PROGRAM Test
VAR
	EdgeD: R_TRIG;
	RS_0: RS;
	CTU_0: CTUD;
	COUNT: CTUD;
	testVar1 : WORD := 11;
	testVar2 : WORD := 0;
	testVar3 : WORD := 12;
		testVar4 : BOOL := TRUE;
		TP_0: TP;
	testVar5 : TIME := T#0ms;
	LEDUBlue: BOOL;
	ms: TIME;
	T1: TON;
	TOF_0: TOF;
	LLBButton: BOOL;
	LED: MotorControla;
	MotorControla_0: MotorControla;
	MotorControla_1: MotorControla;
	MotorControla_2: MotorControla;
	MX: Multiplex;
	Patch: MotorControla;
	MotorControla_3: MotorControla;
	MotorControla_4: MotorControla;
	MotorControla_5: MotorControla;
	IntLck: BOOL;
	IntLck1: BOOL;
	IntLck2: BOOL;
	IntLck3: BOOL;
	Stp3: BOOL;
	Stp1: BOOL;
	Stp2: BOOL;
	Stp4: BOOL;
	Counter_0: Counter;
	KDP: BOOL;
	IntLck4: BOOL;
END_VAR

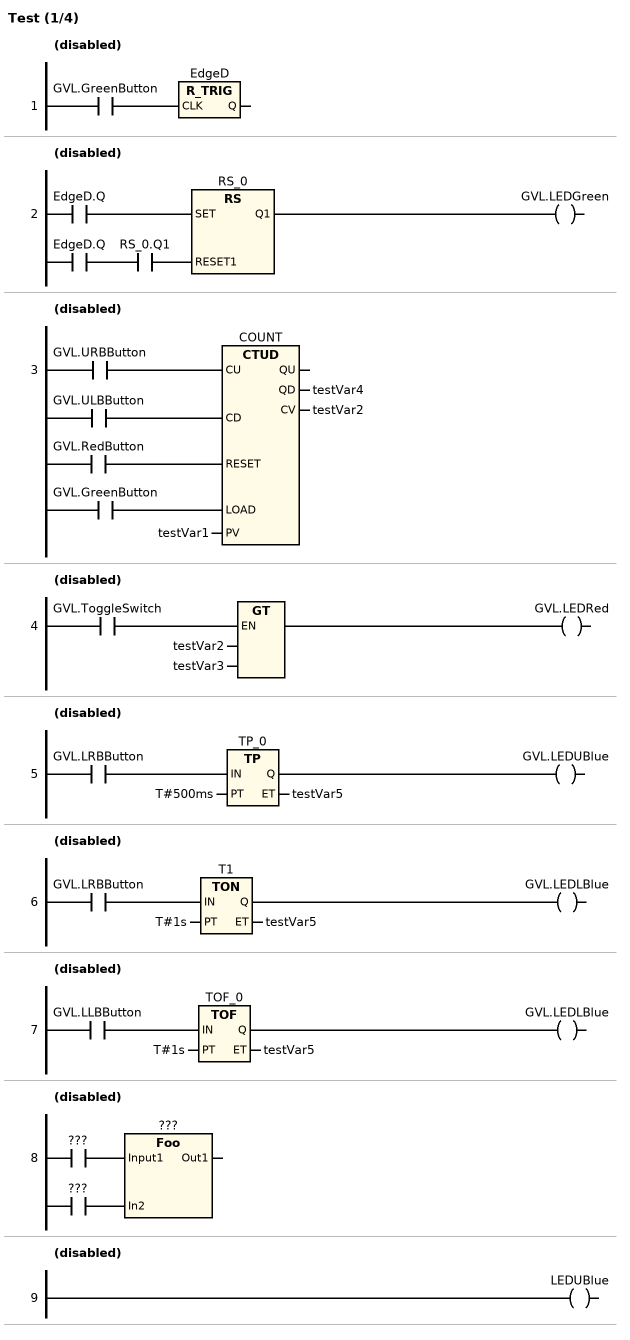
// NETWORK 1 (disabled)
// EdgeD(CLK := GVL.GreenButton); // R_TRIG

// NETWORK 2 (disabled)
// RS_0(SET := EdgeD.Q, RESET1 := EdgeD.Q AND RS_0.Q1); // RS
// GVL.LEDGreen := RS_0.Q1;

// NETWORK 3 (disabled)
// COUNT(
//     CU := GVL.URBButton,
//     CD := GVL.ULBButton,
//     RESET := GVL.RedButton,
//     LOAD := GVL.GreenButton,
//     PV := testVar1,
//     QD => testVar4,
//     CV => testVar2); // CTUD

// NETWORK 4 (disabled)
// GVL.LEDRed := GVL.ToggleSwitch AND testVar2 > testVar3;

// NETWORK 5 (disabled)
// TP_0(IN := GVL.LRBButton, PT := T#500ms, ET => testVar5); // TP
// GVL.LEDUBlue := TP_0.Q;

// NETWORK 6 (disabled)
// T1(IN := GVL.LRBButton, PT := T#1s, ET => testVar5); // TON
// GVL.LEDLBlue := T1.Q;

// NETWORK 7 (disabled)
// TOF_0(IN := GVL.LLBButton, PT := T#1s, ET => testVar5); // TOF
// GVL.LEDLBlue := TOF_0.Q;

// NETWORK 8 (disabled)
// ???(); // Foo

// NETWORK 9 (disabled)
// LEDUBlue := TRUE;

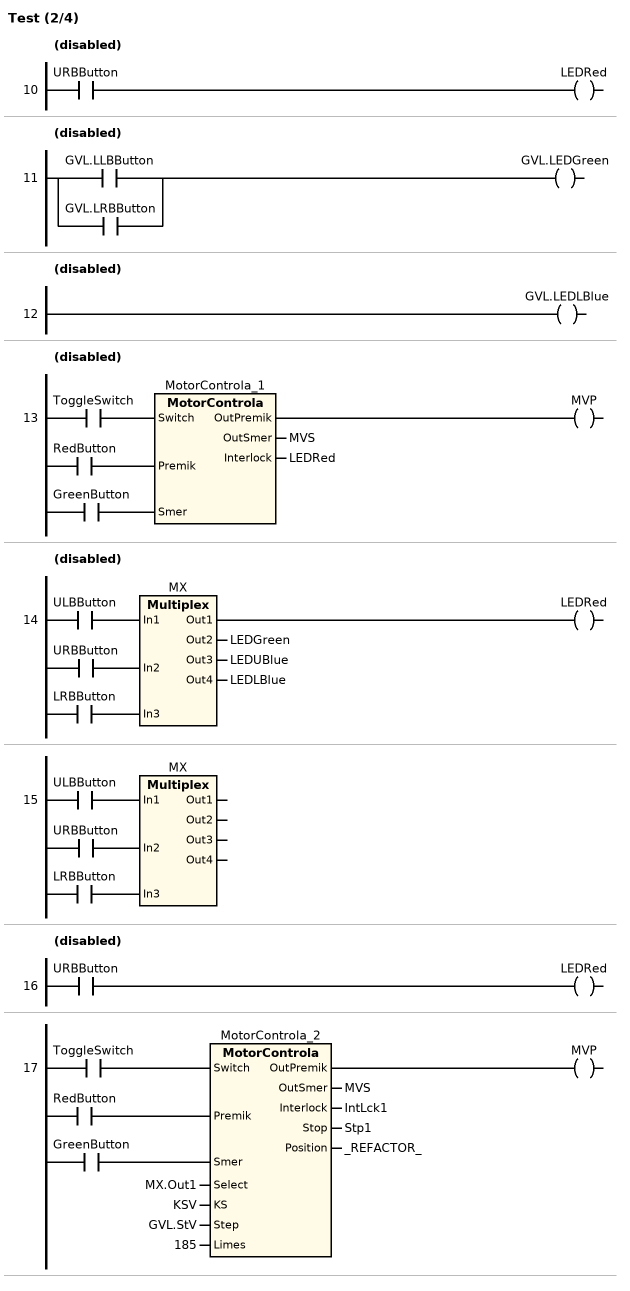
// NETWORK 10 (disabled)
// LEDRed := URBButton;

// NETWORK 11 (disabled)
// GVL.LEDGreen := GVL.LLBButton OR GVL.LRBButton;

// NETWORK 12 (disabled)
// GVL.LEDLBlue := TRUE;

// NETWORK 13 (disabled)
// MotorControla_1(
//     Switch := ToggleSwitch,
//     Premik := RedButton,
//     Smer := GreenButton,
//     OutSmer => MVS,
//     Interlock => LEDRed); // MotorControla
// MVP := MotorControla_1.OutPremik;

// NETWORK 14 (disabled)
// MX(
//     In1 := ULBButton,
//     In2 := URBButton,
//     In3 := LRBButton,
//     Out2 => LEDGreen,
//     Out3 => LEDUBlue,
//     Out4 => LEDLBlue); // Multiplex
// LEDRed := MX.Out1;

// NETWORK 15
MX(In1 := ULBButton, In2 := URBButton, In3 := LRBButton); // Multiplex

// NETWORK 16 (disabled)
// LEDRed := URBButton;

// NETWORK 17
MotorControla_2(
    Switch := ToggleSwitch,
    Premik := RedButton,
    Smer := GreenButton,
    Select := MX.Out1,
    KS := KSV,
    Step := GVL.StV,
    Limes := 185,
    OutSmer => MVS,
    Interlock => IntLck1,
    Stop => Stp1,
    Position => _REFACTOR_); // MotorControla
MVP := MotorControla_2.OutPremik;

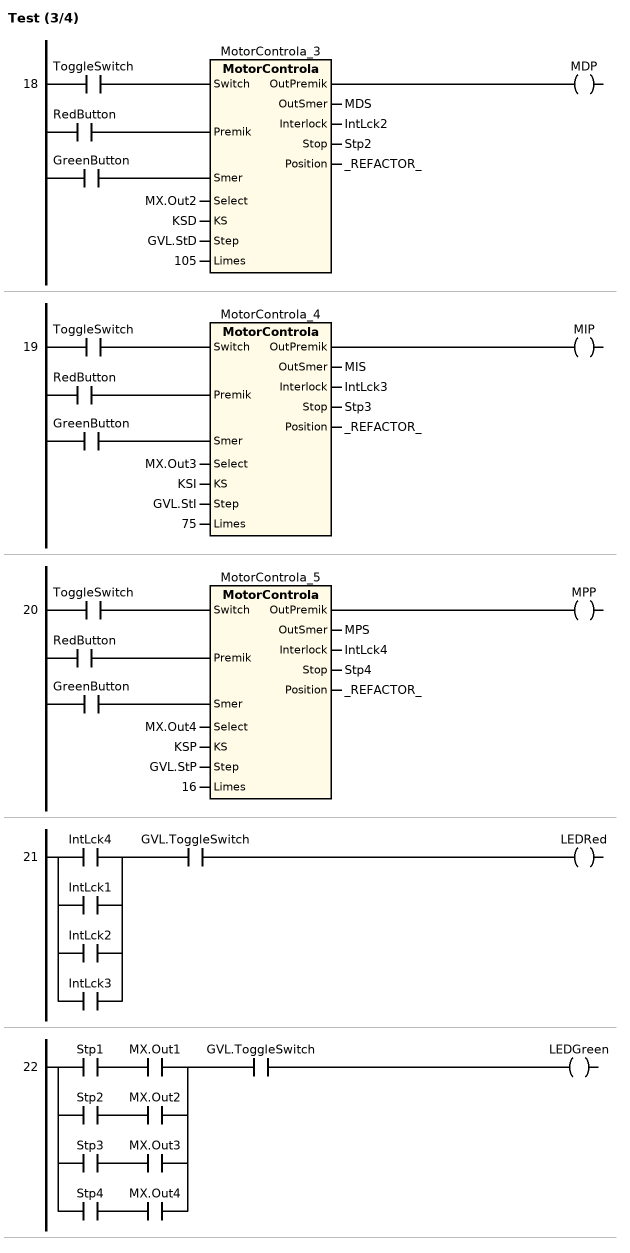
// NETWORK 18
MotorControla_3(
    Switch := ToggleSwitch,
    Premik := RedButton,
    Smer := GreenButton,
    Select := MX.Out2,
    KS := KSD,
    Step := GVL.StD,
    Limes := 105,
    OutSmer => MDS,
    Interlock => IntLck2,
    Stop => Stp2,
    Position => _REFACTOR_); // MotorControla
MDP := MotorControla_3.OutPremik;

// NETWORK 19
MotorControla_4(
    Switch := ToggleSwitch,
    Premik := RedButton,
    Smer := GreenButton,
    Select := MX.Out3,
    KS := KSI,
    Step := GVL.StI,
    Limes := 75,
    OutSmer => MIS,
    Interlock => IntLck3,
    Stop => Stp3,
    Position => _REFACTOR_); // MotorControla
MIP := MotorControla_4.OutPremik;

// NETWORK 20
MotorControla_5(
    Switch := ToggleSwitch,
    Premik := RedButton,
    Smer := GreenButton,
    Select := MX.Out4,
    KS := KSP,
    Step := GVL.StP,
    Limes := 16,
    OutSmer => MPS,
    Interlock => IntLck4,
    Stop => Stp4,
    Position => _REFACTOR_); // MotorControla
MPP := MotorControla_5.OutPremik;

// NETWORK 21
LEDRed := (IntLck4 OR IntLck1 OR IntLck2 OR IntLck3) AND GVL.ToggleSwitch;

// NETWORK 22
LEDGreen := (Stp1 AND MX.Out1 OR Stp2 AND MX.Out2 OR Stp3 AND MX.Out3 OR Stp4 AND MX.Out4) AND GVL.ToggleSwitch;

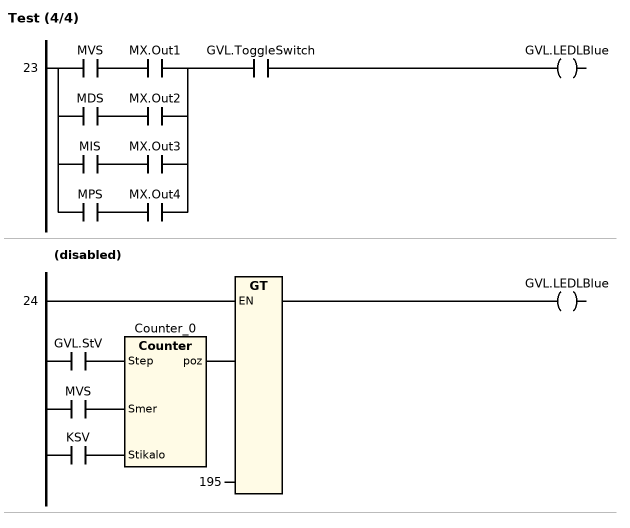
// NETWORK 23
GVL.LEDLBlue := (MVS AND MX.Out1 OR MDS AND MX.Out2 OR MIS AND MX.Out3 OR MPS AND MX.Out4) AND GVL.ToggleSwitch;

// NETWORK 24 (disabled)
// Counter_0(Step := GVL.StV, Smer := MVS, Stikalo := KSV); // Counter
// GVL.LEDLBlue := Counter_0.poz > 195;

END_PROGRAM

(* stored: Version 1.1.0.1, ProductVersion 3.1.4024.12
   POU Test: Id {6726b890-90e1-4c33-ad16-27d2cf874f8b}, SpecialFunc None *)
